(* IEC 61131-3 sources: ATCMcontrol_Engineering/src/TargetBase/Libs/ATCM_Utility2, 25 files *)

(* ---- CloseDB.st ---- *)
(*[[
    UserURL= "CloseDB.htm"
]]*)
FUNCTION CloseDB:DWORD
VAR_INPUT
	DbHandle	: DINT;
	DbType 		: INT;
END_VAR

inline { STDLIB(READDB) }

END_FUNCTION

(* ---- CopyDB.st ---- *)
(*[[
    UserURL= "CopyDB.htm"
]]*)
FUNCTION CopyDB:DWORD
VAR_INPUT
	SourceDbName 	: STRING;
	SourceDbType 	: INT;
	DestDbName 		: STRING;
	DestDbType 		: INT;
	Mode 			: INT;
END_VAR

inline { STDLIB(COPYDB) }

END_FUNCTION

(* ---- CpuUsage.ST ---- *)
(*[[
    UserURL= "CpuUsage.htm"
]]*)

FUNCTION CpuUsage:DWORD

VAR_OUTPUT

   CpuUsePercentage:         UINT;

END_VAR

inline { STDLIB(CPUUSAGE) }

END_FUNCTION

(* ---- CreateDB.st ---- *)
(*[[
    UserURL= "CreateDB.htm"
]]*)
FUNCTION CreateDB:DWORD
VAR_INPUT
	VarName 	: STRING;
	RecordsNum 	: INT;
	DbName 		: STRING;
	DbType 		: INT;
	Mode 		: INT;
END_VAR

inline { STDLIB(CREATEDB) }

END_FUNCTION

(* ---- DeleteDB.st ---- *)
(*[[
    UserURL= "DeleteDB.htm"
]]*)
FUNCTION DeleteDB:DWORD
VAR_INPUT
	DbName 		: STRING;
	DbType 		: INT;
END_VAR

inline { STDLIB(DELETEDB) }

END_FUNCTION

(* ---- FileListDB.st ---- *)
(*[[
    UserURL= "FileListDB.htm"
]]*)
FUNCTION FileListDB:DWORD

VAR_IN_OUT
	DbNamesList	: array of string;
END_VAR

VAR_INPUT
	MaxRecordsNum 	: INT;
	DbType 			: INT;
END_VAR

VAR_OUTPUT
	RecordsNum 	: INT;
END_VAR

inline { STDLIB(FILELISTDB) }

END_FUNCTION

(* ---- ForceRemapInput.st ---- *)
(*[[
    UserURL= "ForceRemapInput.htm"
]]*)
FUNCTION ForceRemapInput:DWORD
VAR_INPUT
	RemapStruct: InRemapStructType;
END_VAR

inline { STDLIB(FORCEREMAPINPUT) }

END_FUNCTION

(* ---- ForceRemapOutput.st ---- *)
(*[[
    UserURL= "ForceRemapOutput.htm"
]]*)
FUNCTION ForceRemapOutput:DWORD
VAR_INPUT
	RemapStruct: OutRemapStructType;
END_VAR

inline { STDLIB(FORCEREMAPOUTPUT) }

END_FUNCTION

(* ---- FreeLibrary.st ---- *)
(*[[
    UserURL= "FreeLibrary.htm",
]]*)

FUNCTION FreeLibrary:DWORD

VAR_INPUT
   LibraryName      : STRING;
END_VAR

inline { STDLIB(FREELIBRARY) }

END_FUNCTION

(* ---- GetDate.ST ---- *)
(*[[
    UserURL= "GetDate.htm"
]]*)

FUNCTION GetDate:DWORD

VAR_OUTPUT

   Day:         ANY_ELEMENTARY;
   Month:       ANY_ELEMENTARY;
   Year:        ANY_ELEMENTARY;
   DayOfWeek:   ANY_ELEMENTARY;

END_VAR

overload DWORD(INT,INT,INT,INT) inline { STDLIB(GETDATE) }
overload DWORD(WORD,WORD,WORD,WORD) inline { STDLIB(GETDATE) }

END_FUNCTION

(* ---- GetTime.ST ---- *)
(*[[
    UserURL= "GetTime.htm",
]]*)

FUNCTION GetTime:DWORD

VAR_OUTPUT

   Hour:       ANY_ELEMENTARY;
   Minute:     ANY_ELEMENTARY;
   Second:     ANY_ELEMENTARY;
   MilliSec:   ANY_ELEMENTARY;

END_VAR

overload DWORD(INT,INT,INT,INT) inline { STDLIB(GETTIME) }
overload DWORD(WORD,WORD,WORD,WORD) inline { STDLIB(GETTIME) }

END_FUNCTION

(* ---- LoadLibrary.st ---- *)
(*[[
    UserURL= "LoadLibrary.htm",
]]*)

FUNCTION LoadLibrary:DWORD

VAR_INPUT
   LibraryName      : STRING;
   StartFunctionOrd : INT;
   EndFunctionOrd   : INT;
   StartFBOrd       : INT;
   EndFBOrd         : INT;
END_VAR

inline { STDLIB(LOADLIBRARY) }

END_FUNCTION

(* ---- OpenDB.st ---- *)
(*[[
    UserURL= "OpenDB.htm"
]]*)
FUNCTION OpenDB:DWORD
VAR_INPUT
	DbName		: STRING;
	DbType		: INT;
END_VAR

VAR_OUTPUT
	DbHandle 	: DINT;
END_VAR

inline { STDLIB(OPENDB) }

END_FUNCTION

(* ---- PurgeRetainDB.st ---- *)
(*[[
    UserURL= "PurgeRetainDB.htm"
]]*)
FUNCTION PurgeRetainDB:DWORD

inline { STDLIB(PURGERETAINDB) }

END_FUNCTION

(* ---- ReadDB.st ---- *)
(*[[
    UserURL= "ReadDB.htm"
]]*)
FUNCTION ReadDB:DWORD
VAR_INPUT
	VarName 	: STRING;
	RecordNum 	: INT;
	DbHandle	: DINT;
	DbType 		: INT;
	Mode 		: INT;
END_VAR

inline { STDLIB(READDB) }

END_FUNCTION

(* ---- ReadRemapInputCFG.st ---- *)
(*[[
    UserURL= "ReadRemapInputCFG.htm"
]]*)

FUNCTION ReadRemapInputCFG:DWORD
VAR_INPUT
	Filename: STRING;
END_VAR

inline { STDLIB(READREMAPINPUTCFG) }

END_FUNCTION

(* ---- ReadRemapOutputCFG.st ---- *)
(*[[
    UserURL= "ReadRemapOutputCFG.htm"
]]*)

FUNCTION ReadRemapOutputCFG:DWORD
VAR_INPUT
	Filename: STRING;
END_VAR

inline { STDLIB(READREMAPOUTPUTCFG) }

END_FUNCTION

(* ---- RemapInput.st ---- *)
(*[[
    UserURL= "RemapInput.htm"
]]*)
FUNCTION RemapInput:DWORD
VAR_INPUT
END_VAR

inline { STDLIB(REMAPINPUT) }

END_FUNCTION

(* ---- RemapOutput.st ---- *)
(*[[
    UserURL= "RemapOutput.htm"
]]*)
FUNCTION RemapOutput:DWORD
VAR_INPUT
END_VAR

inline { STDLIB(REMAPOUTPUT) }

END_FUNCTION

(* ---- RenameDB.st ---- *)
(*[[
    UserURL= "RenameDB.htm"
]]*)
FUNCTION RenameDB:DWORD
VAR_INPUT
	CurrDbName 	: STRING;
	NewDbName 	: STRING;
	DbType 		: INT;
END_VAR

inline { STDLIB(RENAMEDB) }

END_FUNCTION

(* ---- ResizeDB.st ---- *)
(*[[
    UserURL= "ResizeDB.htm"
]]*)
FUNCTION ResizeDB:DWORD
VAR_INPUT
	DbName 			: STRING;
	DbType 			: INT;
	NewRecordsNum 	: INT;
END_VAR

inline { STDLIB(RESIZEDB) }

END_FUNCTION

(* ---- SetDate.ST ---- *)
(*[[
    UserURL= "SetDate.htm",
]]*)

FUNCTION SetDate:DWORD

VAR_INPUT

   Day:       ANY_ELEMENTARY;
   Month:     ANY_ELEMENTARY;
   Year:      ANY_ELEMENTARY;

END_VAR

overload DWORD(INT,INT,INT) inline { STDLIB(SETDATE) }
overload DWORD(WORD,WORD,WORD) inline { STDLIB(SETDATE) }

END_FUNCTION

(* ---- SetTime.ST ---- *)
(*[[
    UserURL= "SetTime.htm",
]]*)

FUNCTION SetTime:DWORD

VAR_INPUT

   Hour:       ANY_ELEMENTARY;
   Minute:     ANY_ELEMENTARY;
   Second:     ANY_ELEMENTARY;
   MilliSec:   ANY_ELEMENTARY;

END_VAR

overload DWORD(INT,INT,INT,INT) inline { STDLIB(SETTIME) }
overload DWORD(WORD,WORD,WORD,WORD) inline { STDLIB(SETTIME) }

END_FUNCTION

(* ---- WriteDB.st ---- *)
(*[[
    UserURL= "WriteDB.htm"
]]*)
FUNCTION WriteDB:DWORD
VAR_INPUT
	VarName 	: STRING;
	RecordNum 	: INT;
	DbHandle	: DINT;
	DbType 		: INT;
	Mode 		: INT;
END_VAR

inline { STDLIB(WRITEDB) }

END_FUNCTION

(* ---- RunProgram.st ---- *)
(*[[
    UserURL= "RunProgram.htm",
]]*)
FUNCTION RunProgram:DWORD
VAR_INPUT
   ExecMode:    INT;
   ProgramName: STRING;
   CommandLine: STRING;
   Timeout:     UDINT; (* expressed in ms *)
END_VAR

inline { STDLIB(RUNPROGRAM) }

END_FUNCTION
